{attribute 'linkalways'} 
{attribute 'no_explicit_call' := 'This FB is a CLASS and must be accessed using methods or properties'}
{attribute 'enable_dynamic_creation'}
FUNCTION_BLOCK Node_F_VN_MinElementElementwise_INT EXTENDS VisionNode
VAR
    ipContainer : _ITcVnContainer;
    nMin : _INT(0);
    hrPrev : _HRESULT(S_OK);
    hresult : _HRESULT(S_OK);
END_VAR

METHOD PUBLIC  Clone : I_Node
VAR
	pNode : POINTER TO Node_F_VN_MinElementElementwise_INT;
END_VAR
pNode := __NEW(Node_F_VN_MinElementElementwise_INT);
Clone := pNode^;
END_METHOD

METHOD FB_init : BOOL
VAR_INPUT
	bInitRetains : BOOL; // if TRUE, the retain variables are initialized (warm start / cold start)
	bInCopyCode : BOOL;  // if TRUE, the instance afterwards gets moved into the copy code (online change)
END_VAR
AddInput('ipContainer', ipContainer);
AddInput('hrPrev', hrPrev);
AddOutput('ipContainer', ipContainer);
AddOutput('nMin', nMin);
AddOutput('hresult',hresult);
END_METHOD

METHOD PROTECTED OnExecute
hresult.Value := F_VN_MinElementElementwise_INT(
    ipContainer := ipContainer.Value,
    nMin := nMin.Value,
    hrPrev:= hrPrev.Value);
END_METHOD

METHOD PUBLIC PreExecutionCheck
VAR_INPUT
	Check : I_PreExecutionChecks;
END_VAR
Check.IsTrue(ipContainer.IsValid, 'ipContainer must be a valid container');
Check.IsTrue(ipContainer.IsType(TC_GLOBAL_CONST_LIST.ContainerType_Vector_INT), 'ipContainer contains incorrect type');
END_METHOD

END_FUNCTION_BLOCK

(* stored: Version 1.1.0.1, ProductVersion 3.1.4026.13
   POU Node_F_VN_MinElementElementwise_INT: Id {642ac5fc-d1cc-4c4b-93ca-4f5309879049}, SpecialFunc None
   Folder Constructor: Id {15c6da6b-27c8-4969-b5c6-349defbae97b}
   Method Clone: Id {d0700a42-02e1-4209-81d9-09a2cfa857ca}
   Method FB_init: Id {6d018d30-6774-42d0-a306-99748d179274}
   Method OnExecute: Id {eedfa52d-13a9-457c-9776-98a62765cd35}
   Method PreExecutionCheck: Id {f43114ab-89d7-4eb3-a27a-2d66d8480dc3} *)
